TYPE TcaRackFeederStatus :
STRUCT
    ActionDescription : STRING(100);	         
	Safe : BOOL;
END_STRUCT
END_TYPE

(* stored: Version 1.1.0.1
   DUT TcaRackFeederStatus: Id {895aba99-7a36-4413-bebb-00d29f85b80f} *)
